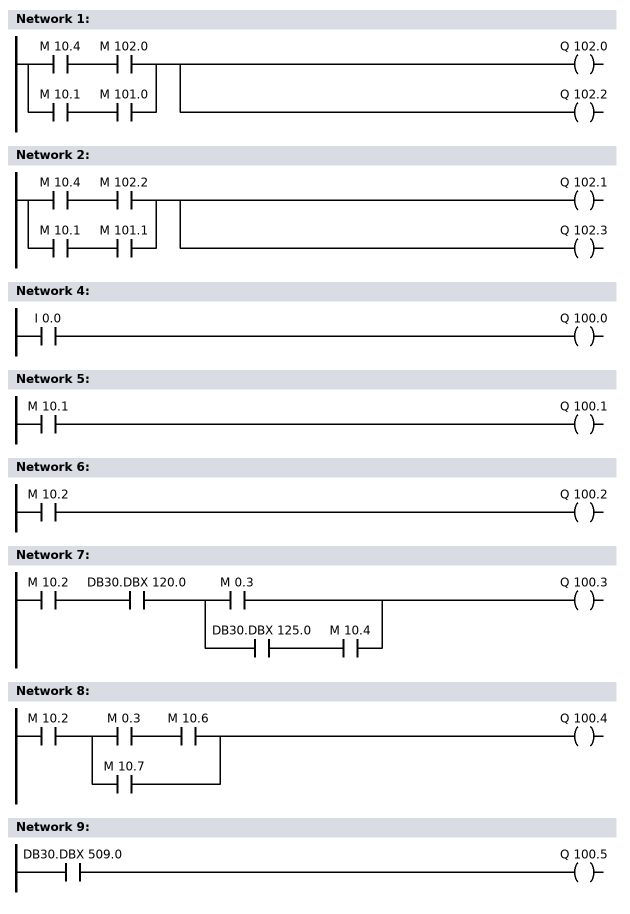
NETWORK
TITLE =
      A     M 10.4;
      A     M 102.0;
      O;
      A     M 10.1;
      A     M 101.0;
      =     Q 102.0;
      =     Q 102.2;
NETWORK
TITLE =
      A     M 10.4;
      A     M 102.2;
      O;
      A     M 10.1;
      A     M 101.1;
      =     Q 102.1;
      =     Q 102.3;
NETWORK
TITLE =
NETWORK
TITLE =
      A     I 0.0;
      =     Q 100.0;
NETWORK
TITLE =
      A     M 10.1;
      =     Q 100.1;
NETWORK
TITLE =
      A     M 10.2;
      =     Q 100.2;
NETWORK
TITLE =
      A     M 10.2;
      A     DB30.DBX 120.0;
      A(;
      O     M 0.3;
      O;
      A     DB30.DBX 125.0;
      A     M 10.4;
      );
      =     Q 100.3;
NETWORK
TITLE =
      A     M 10.2;
      A(;
      A     M 0.3;
      A     M 10.6;
      O     M 10.7;
      );
      =     Q 100.4;
NETWORK
TITLE =
      A     DB30.DBX 509.0;
      =     Q 100.5;
END_FUNCTION

// DB 7: know-how protected block, not included

DATA_BLOCK DB 10
VERSION : 0.1
BEGIN
// 418 bytes; values not shown
END_DATA_BLOCK

DATA_BLOCK DB 15
AUTHOR : AuD_MCE8
FAMILY : FM357_2
NAME : BF_DB15
VERSION : 2.1
FB 6
BEGIN
END_DATA_BLOCK

// DB 16: know-how protected block, not included

// DB 17: know-how protected block, not included

// DB 19: know-how protected block, not included

// DB 20: know-how protected block, not included

DATA_BLOCK DB 21
AUTHOR : AuD_MCE8
FAMILY : FM357_2
NAME : HT6_IF
VERSION : 3.0
BEGIN
// 30 bytes; values not shown
END_DATA_BLOCK

DATA_BLOCK DB 30
VERSION : 0.1
UDT 1
BEGIN
END_DATA_BLOCK

DATA_BLOCK DB 31
VERSION : 0.1
UDT 2
BEGIN
END_DATA_BLOCK

DATA_BLOCK DB 41
VERSION : 0.1
BEGIN
// 2 bytes; values not shown
END_DATA_BLOCK

DATA_BLOCK DB 50
VERSION : 0.1
BEGIN
// 34 bytes; values not shown
END_DATA_BLOCK

DATA_BLOCK DB 60
VERSION : 0.1
BEGIN
// 962 bytes; values not shown
END_DATA_BLOCK

DATA_BLOCK DB 61
VERSION : 0.1
BEGIN
// 500 bytes; values not shown
END_DATA_BLOCK

DATA_BLOCK DB 100
VERSION : 0.1
BEGIN
// 124 bytes; values not shown
END_DATA_BLOCK

DATA_BLOCK DB 105
VERSION : 0.0
BEGIN
// 148 bytes; values not shown
END_DATA_BLOCK

DATA_BLOCK DB 106
AUTHOR : AuD_MCE8
FAMILY : FM357_2
VERSION : 0.0
FB 2
BEGIN
END_DATA_BLOCK

DATA_BLOCK DB 107
AUTHOR : AuD_MCE8
FAMILY : FM357_2
VERSION : 0.0
FB 3
BEGIN
END_DATA_BLOCK

DATA_BLOCK DB 108
VERSION : 0.1
BEGIN
// 200 bytes; values not shown
END_DATA_BLOCK

DATA_BLOCK DB 110
VERSION : 0.1
BEGIN
// 612 bytes; values not shown
END_DATA_BLOCK

DATA_BLOCK DB 115
AUTHOR : AuD_MCE8
FAMILY : FM357_2
NAME : USERDB
VERSION : 3.1
BEGIN
// 130 bytes; values not shown
END_DATA_BLOCK

DATA_BLOCK DB 121
AUTHOR : AuD_MCE8
FAMILY : FM357_2
NAME : VAR_ADDR
VERSION : 3.1
BEGIN
// 190 bytes; values not shown
END_DATA_BLOCK

ORGANIZATION_BLOCK OB 1
VERSION : 1.0
BEGIN
// (block stored without names or comments; labels and parameter names are numbered)
NETWORK
TITLE =
      CALL  FC 22 (
           $1                       := 30);
      A     DB30.DBX 11.0;
      =     DB30.DBX 11.1;
      AN    DB30.DBX 11.1;
      =     M 250.0;
      CALL  FC 21 (
           $1                       := 30,
           $2                       := P#M 250.0,
           $3                       := P#M 252.0);
      A     DB30.DBX 10.2;
      JC    M001;
      A     DB30.DBX 11.1;
      JC    M001;
      CALL  FC 101;
      CALL  FC 102;
M001: NOP   0;
      CALL  FC 100;
NETWORK
TITLE =
      CALL  FC 110;
      CALL  FC 140;
      CALL  FC 160;
      CALL  FC 170;
      CALL  FC 180;
      CALL  FC 190;
      CALL  FC 200;
      CALL  FC 104;
      A     DB30.DBX 108.7;
      =     Q 2.0;
      BE;
END_ORGANIZATION_BLOCK

ORGANIZATION_BLOCK OB 82
VERSION : 1.0
BEGIN
// (block stored without names or comments; labels and parameter names are numbered)
NETWORK
TITLE =
      CALL  FC 5 (
           $1                       := 30);
      BE;
END_ORGANIZATION_BLOCK

ORGANIZATION_BLOCK OB 86
VERSION : 1.1
BEGIN
// (block stored without names or comments; labels and parameter names are numbered)
NETWORK
TITLE =
      L     LB 1;
      L     B#16#C4;
      <>I;
      JC    M004;
      L     LB 11;
      L     B#16#1;
      <>I;
      JC    M003;
      L     B#16#39;
      L     LB 0;
      ==I;
      JC    M001;
      L     B#16#38;
      ==I;
      JC    M002;
      JU    M004;
M001: CALL  FC 5 (
           $1                       := 30);
      JU    M004;
M002: CALL  FC 1 (
           $1                       := 30,
           $2                       := 256,
           $3                       := 100,
           $4                       := TRUE,
           $5                       := TRUE);
      JU    M004;
M003: NOP   0;
M004: BE;
END_ORGANIZATION_BLOCK

ORGANIZATION_BLOCK OB 87
VERSION : 0.1
BEGIN
// (block stored without names or comments; labels and parameter names are numbered)
END_ORGANIZATION_BLOCK

ORGANIZATION_BLOCK OB 100
VERSION : 1.0
BEGIN
// (block stored without names or comments; labels and parameter names are numbered)
NETWORK
TITLE =
      CALL  FC 1 (
           $1                       := 30,
           $2                       := 256,
           $3                       := 100,
           $4                       := TRUE,
           $5                       := TRUE);
      BE;
END_ORGANIZATION_BLOCK

ORGANIZATION_BLOCK OB 121
VERSION : 0.1
BEGIN
// (block stored without names or comments; labels and parameter names are numbered)
END_ORGANIZATION_BLOCK

ORGANIZATION_BLOCK OB 122
VERSION : 0.1
BEGIN
// (block stored without names or comments; labels and parameter names are numbered)
END_ORGANIZATION_BLOCK
